INTERFACE I_HE_SolidAttenuatorFilter EXTENDS I_Fallible


METHOD GetCenterPosition
VAR_INPUT
    CenterPosition : I_QuantityLREALPublic;
END_VAR
END_METHOD


METHOD GetLength
VAR_INPUT
    Length : I_QuantityLREALPublic;
END_VAR
END_METHOD


METHOD GetMaterial
VAR_IN_OUT
    Material : T_MaxString;
END_VAR
END_METHOD


METHOD GetThicknessAt
VAR_INPUT
    QueryPointInAxisCoordinates : I_QuantityLREAL;
    Thickness : I_QuantityLREALPublic;
END_VAR
END_METHOD

END_INTERFACE

(* stored: Version 1.1.0.1
   Itf I_HE_SolidAttenuatorFilter: Id {032eac1f-d222-4245-a784-ead19447a336}
   Method GetCenterPosition: Id {731d3cdb-270e-4cff-906f-e5973c584cf9}
   Method GetLength: Id {09e64b52-ce20-4c07-9046-9f95ec96daa5}
   Method GetMaterial: Id {01627194-3c3f-4ca7-bdaf-b6736b4f8407}
   Method GetThicknessAt: Id {bb7b6406-6e35-4c8c-847b-171628725a98} *)
